(* PLC project test_ethercat, Laurent BESSARD test_ethercat 1.0 *)
(* stored: creationDateTime 2011-10-20T19:01:52, modificationDateTime 2012-02-15T00:53:41 *)

PROGRAM Prog
  VAR
    CLOCK AT %QX0.0.0.2.28672.1 : BOOL;
    LED AT %QX0.0.0.2.28688.1 : BOOL := TRUE;
    ControlWord AT %QW0.0.1.0.24640.0 : UINT;
    StatusWord AT %IW0.0.1.0.24641.0 : UINT;
    ErrorCode AT %IW0.0.1.0.24639.0 : UINT;
    Mode AT %IB0.0.1.0.24673.0 : SINT;
  END_VAR

CLOCK := NOT CLOCK;
          
END_PROGRAM

CONFIGURATION conf
  RESOURCE res ON PLC
    TASK main_task(INTERVAL := T#0.4ms, PRIORITY := 0);
    PROGRAM main_instance WITH main_task : Prog;
  END_RESOURCE
END_CONFIGURATION
